(* PLC project door, Dassault Systèmes ControlBuild 2024x *)
(* stored: creationDateTime 2023-10-03T11:13:52-01:00 *)

PROGRAM tni_train.door
  VAR_INPUT
    compressedAir : REAL := 200.0;
    cmdSupply : BOOL := true;
    sensorSupply : BOOL := true;
  END_VAR
  VAR_INPUT
    enableOpening : BOOL := false;
    enableClosing : BOOL := false;
  END_VAR
  VAR_OUTPUT
    closedDoorState : BOOL := false;
    openedDoorState : BOOL := false;
    faultState : DINT := 0;
  END_VAR

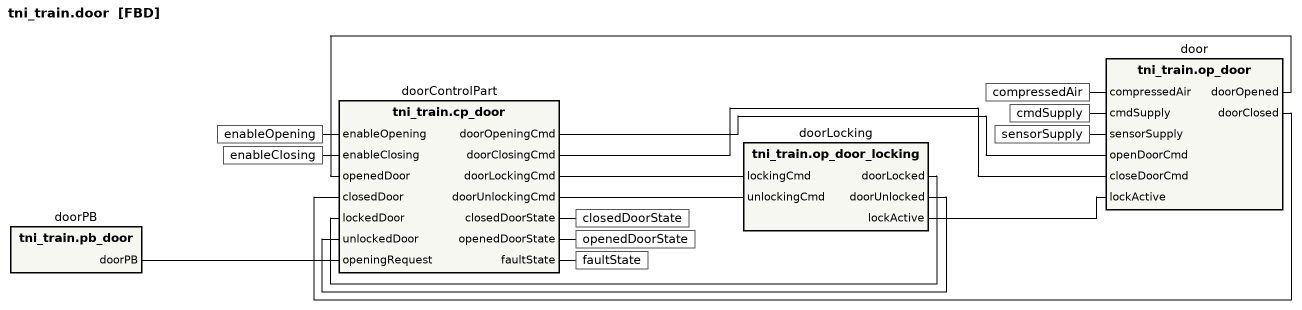
(* FBD diagram, written out as Structured Text *)
doorLocking(lockingCmd := doorControlPart.doorLockingCmd, unlockingCmd := doorControlPart.doorUnlockingCmd);
door(compressedAir := compressedAir, cmdSupply := cmdSupply, sensorSupply := sensorSupply, openDoorCmd := doorControlPart.doorOpeningCmd, closeDoorCmd := doorControlPart.doorClosingCmd, lockActive := doorLocking.lockActive);
doorPB();
doorControlPart(enableOpening := enableOpening, enableClosing := enableClosing, openedDoor := door.doorOpened, closedDoor := door.doorClosed, lockedDoor := doorLocking.doorLocked, unlockedDoor := doorLocking.doorUnlocked, openingRequest := doorPB.doorPB);
closedDoorState := doorControlPart.closedDoorState;
openedDoorState := doorControlPart.openedDoorState;
faultState := doorControlPart.faultState;
END_PROGRAM
